// TIA Portal V20 export
// export: Created 2026-04-11T06:02:29.8299508Z, ExportSetting WithDefaults, DisplayName Totally Integrated Automation Portal, DisplayVersion V20, DisplayName TIA Portal Openness, DisplayVersion V20, DisplayName TIA Portal Version Control Interface, DisplayVersion V20, DisplayName STEP 7 Professional, DisplayVersion V20, DisplayName STEP 7 Safety, DisplayVersion V20, DisplayName WinCC Basic/Comfort/Advanced, DisplayVersion V20, DisplayName WinCC Unified, DisplayVersion V20
TYPE "udtError_Simocode"
// stored: IsFailsafeCompliant false
   STRUCT
      MotorProtectorTripped { ExternalWritable := 'False'} : Bool;   // Motor protector tripped
      NoSignalForward { ExternalWritable := 'False'} : Bool;   // No signal forward from Simocode
      NoSignalReverse { ExternalWritable := 'False'} : Bool;   // No signal reverse from Simocode (Reversing starter only)
      MotorOverload { ExternalWritable := 'False'} : Bool;   // Motor overload
      GeneralFault { ExternalWritable := 'False'} : Bool;   // Simocode Fault
      NotInRemote { ExternalWritable := 'False'} : Bool;   // Module not in remote mode
      MotorNotStopped { ExternalWritable := 'False'} : Bool;   // Motor doesn't stop
      LocalDisconnectOff { ExternalWritable := 'False'} : Bool;   // Local disconnect off
   END_STRUCT;
END_TYPE
